// TIA Portal project "Automated" (V16)

(* hardware
DEVICE "S7300/ET200M station_1"  S7-300 station
   slot 0: "Rail_0"  Rail  6ES7 390-1***0-0AA0
   slot 2: "PLC_1"  CPU 313C-2 DP  6ES7 313-6CG04-0AB0  V3.3
      slot 0: "MPI interface_1"  MPI
      slot 1: "DP interface_1"  DP
      slot 2: "DI 16/DO 16_1"  DI16/DO16
      slot 4: "Count_1"  Counter
*)

// ===== PLC "PLC_1"  CPU 313C-2 DP =====

VAR_GLOBAL   // PLC tag table "Default tag table"
   "at entry" AT %I0.0 : Bool;
   "at load" AT %I0.1 : Bool;
   "at left" AT %I0.2 : Bool;
   "at middle" AT %I0.3 : Bool;
   "at right" AT %I0.4 : Bool;
   "at unload" AT %I0.5 : Bool;
   "at exit" AT %I0.6 : Bool;
   "moving X" AT %I0.7 : Bool;
   "moving z" AT %I1.0 : Bool;
   "start" AT %I1.1 : Bool;
   "reset" AT %I1.2 : Bool;
   "stop" AT %I1.3 : Bool;
   "entry conveyor" AT %Q0.0 : Bool;
   "load conveyor" AT %Q0.1 : Bool;
   "forks left" AT %Q0.2 : Bool;
   "forks right" AT %Q0.3 : Bool;
   "lift" AT %Q0.4 : Bool;
   "unload conveyor" AT %Q0.5 : Bool;
   "exit conveyor" AT %Q0.6 : Bool;
   "start light" AT %Q0.7 : Bool;
   "reset light" AT %Q1.0 : Bool;
   "stop light" AT %Q1.1 : Bool;
   "target position" AT %QW30 : Int;
   "state0" AT %M0.0 : Bool;
   "state1" AT %M0.1 : Bool;
   "state2" AT %M0.2 : Bool;
   "state3" AT %M0.3 : Bool;
   "state4" AT %M0.4 : Bool;
   "state5" AT %M0.5 : Bool;
   "state6" AT %M0.6 : Bool;
   "state7" AT %M0.7 : Bool;
   "state8" AT %M1.0 : Bool;
   "state9" AT %M1.1 : Bool;
   "Tag_1" AT %M1.2 : Bool;
   "Tag_2" AT %M1.3 : Bool;
   "Tag_3" AT %M1.4 : Bool;
   "Tag_4" AT %M1.5 : Bool;
   "Tag_5" AT %M1.6 : Bool;
   "t" AT %MW30 : Int;
   "Tag_6" AT %M1.7 : Bool;
END_VAR

FUNCTION "Start Stop" : Void   // FC1, LAD
{ S7_Optimized_Access := 'FALSE' }
VERSION : 0.1
BEGIN

REGION Network 1
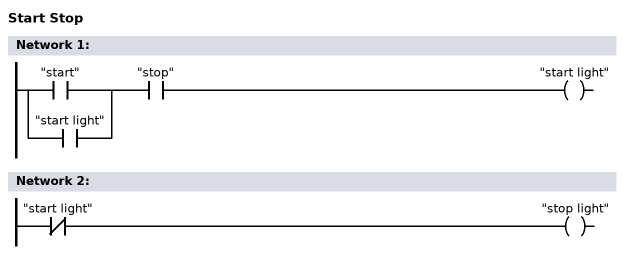
   RUNG wire#powerrail
      Contact( "start" )
      wire#w1
      Contact( "stop" )
      Coil( "start light" )
   END_RUNG
   RUNG wire#powerrail
      Contact( "start light" )
   END_RUNG wire#w1
   // the same network as SCL:
   "start light" := ("start" OR "start light") AND "stop";
END_REGION

REGION Network 2
   RUNG wire#powerrail
      I_Contact( "start light" )
      Coil( "stop light" )
   END_RUNG
   // the same network as SCL:
   "stop light" := NOT "start light";
END_REGION
END_FUNCTION

FUNCTION "State" : Void   // FC2, LAD
{ S7_Optimized_Access := 'FALSE' }
VERSION : 0.1
   VAR_TEMP   // added for the SCL form of the ladder/FBD networks
      _w1 : Bool;
      _w2 : Bool;
   END_VAR
BEGIN

REGION Network 1
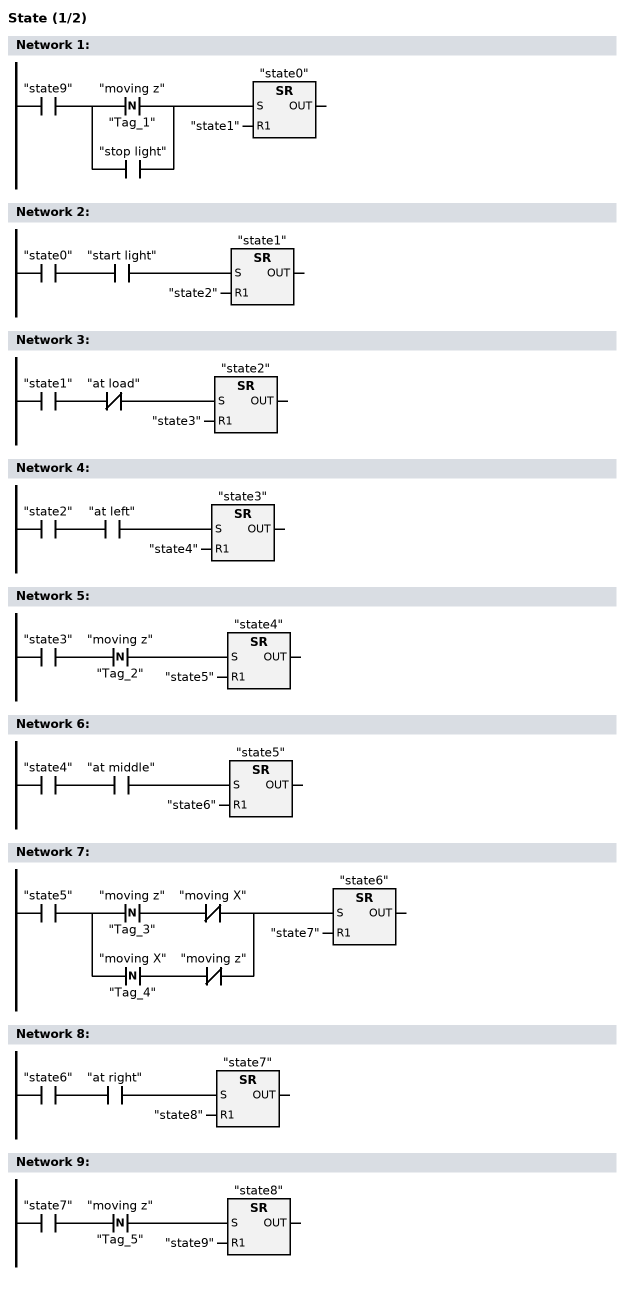
   RUNG wire#powerrail
      Contact( "state9" )
      wire#w1
      N_Contact(operand := "moving z", bit := "Tag_1")
      wire#w2
      S_SR(operand := "state0", r1 := "state1")
   END_RUNG
   RUNG wire#w1
      Contact( "stop light" )
   END_RUNG wire#w2
   // the same network as SCL:
   #_w1 := "state9" AND NOT "moving z" AND "Tag_1";   // falling edge of "moving z"
   "Tag_1" := "moving z";
   IF #_w1 OR ("state9" AND "stop light") THEN
       "state0" := TRUE;   // SR flip-flop
   END_IF;
   IF "state1" THEN "state0" := FALSE; END_IF;
END_REGION

REGION Network 2
   RUNG wire#powerrail
      Contact( "state0" )
      Contact( "start light" )
      S_SR(operand := "state1", r1 := "state2")
   END_RUNG
   // the same network as SCL:
   IF "state0" AND "start light" THEN
       "state1" := TRUE;   // SR flip-flop
   END_IF;
   IF "state2" THEN "state1" := FALSE; END_IF;
END_REGION

REGION Network 3
   RUNG wire#powerrail
      Contact( "state1" )
      I_Contact( "at load" )
      S_SR(operand := "state2", r1 := "state3")
   END_RUNG
   // the same network as SCL:
   IF "state1" AND NOT "at load" THEN
       "state2" := TRUE;   // SR flip-flop
   END_IF;
   IF "state3" THEN "state2" := FALSE; END_IF;
END_REGION

REGION Network 4
   RUNG wire#powerrail
      Contact( "state2" )
      Contact( "at left" )
      S_SR(operand := "state3", r1 := "state4")
   END_RUNG
   // the same network as SCL:
   IF "state2" AND "at left" THEN
       "state3" := TRUE;   // SR flip-flop
   END_IF;
   IF "state4" THEN "state3" := FALSE; END_IF;
END_REGION

REGION Network 5
   RUNG wire#powerrail
      Contact( "state3" )
      N_Contact(operand := "moving z", bit := "Tag_2")
      S_SR(operand := "state4", r1 := "state5")
   END_RUNG
   // the same network as SCL:
   #_w1 := "state3" AND NOT "moving z" AND "Tag_2";   // falling edge of "moving z"
   "Tag_2" := "moving z";
   IF #_w1 THEN
       "state4" := TRUE;   // SR flip-flop
   END_IF;
   IF "state5" THEN "state4" := FALSE; END_IF;
END_REGION

REGION Network 6
   RUNG wire#powerrail
      Contact( "state4" )
      Contact( "at middle" )
      S_SR(operand := "state5", r1 := "state6")
   END_RUNG
   // the same network as SCL:
   IF "state4" AND "at middle" THEN
       "state5" := TRUE;   // SR flip-flop
   END_IF;
   IF "state6" THEN "state5" := FALSE; END_IF;
END_REGION

REGION Network 7
   RUNG wire#powerrail
      Contact( "state5" )
      wire#w1
      N_Contact(operand := "moving z", bit := "Tag_3")
      I_Contact( "moving X" )
      wire#w2
      S_SR(operand := "state6", r1 := "state7")
   END_RUNG
   RUNG wire#w1
      N_Contact(operand := "moving X", bit := "Tag_4")
      I_Contact( "moving z" )
   END_RUNG wire#w2
   // the same network as SCL:
   #_w1 := "state5" AND NOT "moving z" AND "Tag_3";   // falling edge of "moving z"
   "Tag_3" := "moving z";
   #_w2 := "state5" AND NOT "moving X" AND "Tag_4";   // falling edge of "moving X"
   "Tag_4" := "moving X";
   IF (#_w1 AND NOT "moving X") OR (#_w2 AND NOT "moving z") THEN
       "state6" := TRUE;   // SR flip-flop
   END_IF;
   IF "state7" THEN "state6" := FALSE; END_IF;
END_REGION

REGION Network 8
   RUNG wire#powerrail
      Contact( "state6" )
      Contact( "at right" )
      S_SR(operand := "state7", r1 := "state8")
   END_RUNG
   // the same network as SCL:
   IF "state6" AND "at right" THEN
       "state7" := TRUE;   // SR flip-flop
   END_IF;
   IF "state8" THEN "state7" := FALSE; END_IF;
END_REGION

REGION Network 9
   RUNG wire#powerrail
      Contact( "state7" )
      N_Contact(operand := "moving z", bit := "Tag_5")
      S_SR(operand := "state8", r1 := "state9")
   END_RUNG
   // the same network as SCL:
   #_w1 := "state7" AND NOT "moving z" AND "Tag_5";   // falling edge of "moving z"
   "Tag_5" := "moving z";
   IF #_w1 THEN
       "state8" := TRUE;   // SR flip-flop
   END_IF;
   IF "state9" THEN "state8" := FALSE; END_IF;
END_REGION

REGION Network 10
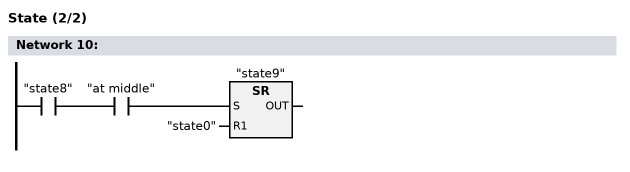
   RUNG wire#powerrail
      Contact( "state8" )
      Contact( "at middle" )
      S_SR(operand := "state9", r1 := "state0")
   END_RUNG
   // the same network as SCL:
   IF "state8" AND "at middle" THEN
       "state9" := TRUE;   // SR flip-flop
   END_IF;
   IF "state0" THEN "state9" := FALSE; END_IF;
END_REGION
END_FUNCTION

FUNCTION "Actuator" : Void   // FC3, LAD
{ S7_Optimized_Access := 'FALSE' }
VERSION : 0.1
   VAR_TEMP   // added for the SCL form of the ladder/FBD networks
      _w1 : Bool;
   END_VAR
BEGIN

REGION Network 1
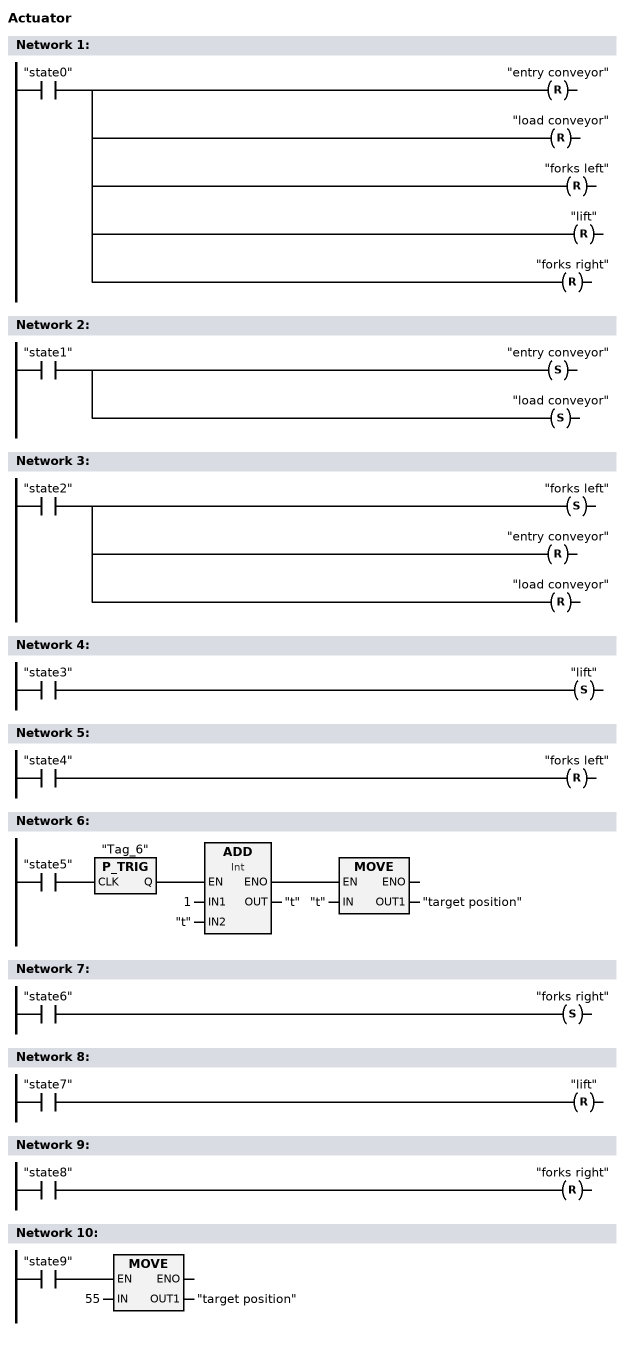
   RUNG wire#powerrail
      Contact( "state0" )
      wire#w1
      R_Coil( "entry conveyor" )
   END_RUNG
   RUNG wire#w1
      R_Coil( "load conveyor" )
   END_RUNG
   RUNG wire#w1
      R_Coil( "forks left" )
   END_RUNG
   RUNG wire#w1
      R_Coil( "lift" )
   END_RUNG
   RUNG wire#w1
      R_Coil( "forks right" )
   END_RUNG
   // the same network as SCL:
   IF "state0" THEN
       "entry conveyor" := FALSE;
       "load conveyor" := FALSE;
       "forks left" := FALSE;
       "lift" := FALSE;
       "forks right" := FALSE;
   END_IF;
END_REGION

REGION Network 2
   RUNG wire#powerrail
      Contact( "state1" )
      wire#w1
      S_Coil( "entry conveyor" )
   END_RUNG
   RUNG wire#w1
      S_Coil( "load conveyor" )
   END_RUNG
   // the same network as SCL:
   IF "state1" THEN
       "entry conveyor" := TRUE;
       "load conveyor" := TRUE;
   END_IF;
END_REGION

REGION Network 3
   RUNG wire#powerrail
      Contact( "state2" )
      wire#w1
      S_Coil( "forks left" )
   END_RUNG
   RUNG wire#w1
      R_Coil( "entry conveyor" )
   END_RUNG
   RUNG wire#w1
      R_Coil( "load conveyor" )
   END_RUNG
   // the same network as SCL:
   IF "state2" THEN
       "forks left" := TRUE;
       "entry conveyor" := FALSE;
       "load conveyor" := FALSE;
   END_IF;
END_REGION

REGION Network 4
   RUNG wire#powerrail
      Contact( "state3" )
      S_Coil( "lift" )
   END_RUNG
   // the same network as SCL:
   IF "state3" THEN "lift" := TRUE; END_IF;
END_REGION

REGION Network 5
   RUNG wire#powerrail
      Contact( "state4" )
      R_Coil( "forks left" )
   END_RUNG
   // the same network as SCL:
   IF "state4" THEN "forks left" := FALSE; END_IF;
END_REGION

REGION Network 6
   RUNG wire#powerrail
      Contact( "state5" )
      P_Trig( "Tag_6" )
      { S7_Templates := "SrcType := Int"; S7_GenerateENO := "TRUE" } Add(in1 := 1, in2 := "t", out => "t")
      { S7_GenerateENO := "TRUE" } Move(in := "t", out1 => "target position")
   END_RUNG
   // the same network as SCL:
   // ENO of a box is taken as its EN; it also drops when the box reports an error
   #_w1 := "state5" AND NOT "Tag_6";   // rising edge
   "Tag_6" := "state5";
   IF #_w1 THEN
       "t" := 1 + "t";
       "target position" := "t";
   END_IF;
END_REGION

REGION Network 7
   RUNG wire#powerrail
      Contact( "state6" )
      S_Coil( "forks right" )
   END_RUNG
   // the same network as SCL:
   IF "state6" THEN "forks right" := TRUE; END_IF;
END_REGION

REGION Network 8
   RUNG wire#powerrail
      Contact( "state7" )
      R_Coil( "lift" )
   END_RUNG
   // the same network as SCL:
   IF "state7" THEN "lift" := FALSE; END_IF;
END_REGION

REGION Network 9
   RUNG wire#powerrail
      Contact( "state8" )
      R_Coil( "forks right" )
   END_RUNG
   // the same network as SCL:
   IF "state8" THEN "forks right" := FALSE; END_IF;
END_REGION

REGION Network 10
   RUNG wire#powerrail
      Contact( "state9" )
      { S7_GenerateENO := "TRUE" } Move(in := 55, out1 => "target position")
   END_RUNG
   // the same network as SCL:
   IF "state9" THEN "target position" := 55; END_IF;
END_REGION
END_FUNCTION

ORGANIZATION_BLOCK "Main"   // OB1, LAD
TITLE = "Main Program Sweep (Cycle)"
{ S7_Optimized_Access := 'FALSE' }
VERSION : 0.1
   VAR_TEMP
      OB1_EV_CLASS : Byte;   // Bits 0-3 = 1 (Coming event), Bits 4-7 = 1 (Event class 1)
      OB1_SCAN_1 : Byte;   // 1 (Cold restart scan 1 of OB 1), 3 (Scan 2-n of OB 1)
      OB1_PRIORITY : Byte;   // Priority of OB Execution
      OB1_OB_NUMBR : Byte;   // 1 (Organization block 1, OB1)
      OB1_RESERVED_1 : Byte;   // Reserved for system
      OB1_RESERVED_2 : Byte;   // Reserved for system
      OB1_PREV_CYCLE : Int;   // Cycle time of previous OB1 scan (milliseconds)
      OB1_MIN_CYCLE : Int;   // Minimum cycle time of OB1 (milliseconds)
      OB1_MAX_CYCLE : Int;   // Maximum cycle time of OB1 (milliseconds)
      OB1_DATE_TIME : Date_And_Time;   // Date and time OB1 started
   END_VAR
BEGIN

REGION Network 1
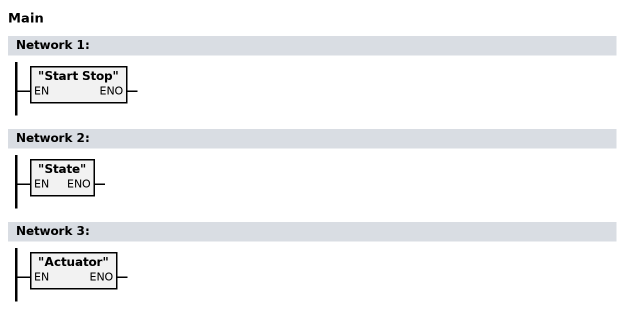
   RUNG wire#powerrail
      "Start Stop"()
   END_RUNG
   // the same network as SCL:
   "Start Stop"();
END_REGION

REGION Network 2
   RUNG wire#powerrail
      "State"()
   END_RUNG
   // the same network as SCL:
   "State"();
END_REGION

REGION Network 3
   RUNG wire#powerrail
      "Actuator"()
   END_RUNG
   // the same network as SCL:
   "Actuator"();
END_REGION
END_ORGANIZATION_BLOCK

ORGANIZATION_BLOCK "COMPLETE RESTART"   // OB100, LAD
TITLE = "Complete Restart"
{ S7_Optimized_Access := 'FALSE' }
VERSION : 0.1
   VAR_TEMP
      OB100_EV_CLASS : Byte;   // 16#13, Event class 1, Entering event state, Event logged in diagnostic buffer
      OB100_STRTUP : Byte;   // 16#81/82/83/84 Method of startup
      OB100_PRIORITY : Byte;   // Priority of OB Execution
      OB100_OB_NUMBR : Byte;   // 100 (Organization block 100, OB100)
      OB100_RESERVED_1 : Byte;   // Reserved for system
      OB100_RESERVED_2 : Byte;   // Reserved for system
      OB100_STOP : Word;   // Event that caused CPU to stop (16#4xxx)
      OB100_STRT_INFO : DWord;   // Information on how system started
      OB100_DATE_TIME : Date_And_Time;   // Date and time OB100 started
   END_VAR
BEGIN

REGION Network 1
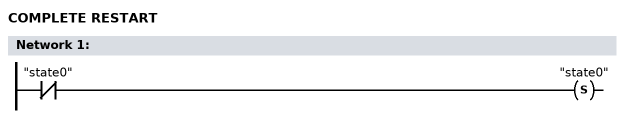
   RUNG wire#powerrail
      I_Contact( "state0" )
      S_Coil( "state0" )
   END_RUNG
   // the same network as SCL:
   IF NOT "state0" THEN "state0" := TRUE; END_IF;
END_REGION
END_ORGANIZATION_BLOCK